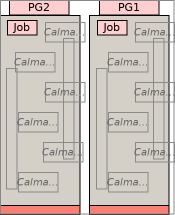
VISUALIZATION _VISU_PmEnable  // 175x215
VAR_IN_OUT
  mInst : FB_PrintModule_Base;
END_VAR
    RoundedRectangle (0,15 80x200), tooltip "Worker enable"
        toggle mInst.fbWorkerPrint[2]._bEnable
    RoundedRectangle (89,15 80x200), tooltip "Worker enable"
        toggle mInst.fbWorkerPrint[1].bWorkerEnable
    Frame (153,38 11x121)
        shows CalmarCompPrint._VISU_PC_MiniVertical(mInst := mInst._pPc[1]^)
    Frame (96,68 11x121)
        shows CalmarCompPrint._VISU_PC_MiniVertical(mInst := mInst._pPc[2]^)
    Frame (135,22 40x20)
        shows CalmarCompPrint._VISU_PH_TinyVertical(mInst := mInst._pPh[1]^)
    Frame (108,52 40x20)
        shows CalmarCompPrint._VISU_PH_TinyVertical(mInst := mInst._pPh[2]^)
    Frame (135,82 40x20)
        shows CalmarCompPrint._VISU_PH_TinyVertical(mInst := mInst._pPh[3]^)
    Frame (108,112 40x20)
        shows CalmarCompPrint._VISU_PH_TinyVertical(mInst := mInst._pPh[4]^)
    Frame (135,142 40x20)
        shows CalmarCompPrint._VISU_PH_TinyVertical(mInst := mInst._pPh[5]^)
    Frame (108,172 40x20)
        shows CalmarCompPrint._VISU_PH_TinyVertical(mInst := mInst._pPh[6]^)
    Frame (63,38 11x121)
        shows CalmarCompPrint._VISU_PC_MiniVertical(mInst := mInst._pPc[3]^)
    Frame (6,68 11x121)
        shows CalmarCompPrint._VISU_PC_MiniVertical(mInst := mInst._pPc[4]^)
    Frame (45,22 40x20)
        shows CalmarCompPrint._VISU_PH_TinyVertical(mInst := mInst._pPh[7]^)
    Frame (15,52 40x20)
        shows CalmarCompPrint._VISU_PH_TinyVertical(mInst := mInst._pPh[8]^)
    Frame (45,82 40x20)
        shows CalmarCompPrint._VISU_PH_TinyVertical(mInst := mInst._pPh[9]^)
    Frame (18,112 40x20)
        shows CalmarCompPrint._VISU_PH_TinyVertical(mInst := mInst._pPh[10]^)
    Frame (43,142 40x20)
        shows CalmarCompPrint._VISU_PH_TinyVertical(mInst := mInst._pPh[11]^)
    Frame (18,172 40x20)
        shows CalmarCompPrint._VISU_PH_TinyVertical(mInst := mInst._pPh[12]^)
    RoundedRectangle (99,0 60x15), "PG1", tooltip "PG: %s"
        p4168582468: mInst.fbWorkerPrint[1]._pAdsPg^.stAds.aO_Name
        toggle mInst.fbWorkerPrint[1]._pAdsPg^.stAds.bI_Enable
    RoundedRectangle (9,0 60x15), "PG2", tooltip "PG: %s"
        p4168582468: mInst.fbWorkerPrint[1]._pAdsPg^.stAds.aO_Name
        toggle mInst.fbWorkerPrint[2]._pAdsPg^.stAds.bI_Enable
    RoundedRectangle (89,205 80x10), tooltip "Worker PrintEnable"
        toggle mInst.fbWorkerPrint[1].bWorkerPrintEnable
    RoundedRectangle (0,205 80x10), tooltip "Worker PrintEnable"
        toggle mInst.fbWorkerPrint[2].bWorkerPrintEnable
    RoundedRectangle (97,20 30x15), "Job", tooltip "Job is active", colour toggle: mInst.fbWorkerPrint[1]._bJobActive
    RoundedRectangle (7,20 30x15), "Job", tooltip "Job is active", colour toggle: mInst.fbWorkerPrint[2]._bJobActive
END_VISUALIZATION

(* stored: Version 1.1.0.1, ProductVersion 3.1.4024.11
   Visu _VISU_PmEnable: Id {df2e315b-c1d5-415d-af8a-9b855c91230b} *)
